TYPE ST_Ti5CiA402PdoOutput :
STRUCT
    nControlword : UINT;
    nModeOfOperation : SINT;
    nTargetPosition : DINT;
    nTargetVelocity : DINT;
END_STRUCT
END_TYPE

(* stored: Version 1.1.0.1, ProductVersion 3.1.4024.0 *)
